{attribute 'qualified_only'}
VAR_GLOBAL
	
	fControlValveSignal : REAL; // -1 - 1 u-signal
	
END_VAR

(* stored: Version 1.1.0.1, ProductVersion 3.1.4024.10
   GVL DigitaloOutput: Id {c0721c33-139a-485f-9d56-3f43f4d2e3ce} *)
